FUNCTION_BLOCK PUBLIC MoveMoverToPositionZoned EXTENDS MoveMoverToPosition
VAR_INPUT
END_VAR
VAR_OUTPUT
END_VAR
VAR
	StartZone: INT;
	CurrentZone : INT;
	ZoneTransitionPositions : ARRAY[1..4] OF LREAL;
	ZoneVelocities : ARRAY[1..4] OF MC_LREAL;
END_VAR

METHOD Cycle : BOOL
VAR_INPUT
END_VAR
CASE State OF
	0:
		IF _MoveMover THEN
			_done := FALSE;
			_error := FALSE;
			_busy := TRUE;
			moveAbs.Execute := TRUE;
			StartZone := GetZone();
			moveAbs.Velocity := ZoneVelocities[StartZone];
			IF moveAbs.Busy THEN
				State := 10;
				_MoveMover := FALSE;
			END_IF
		END_IF
	
	10:
		IF NOT moveAbs.Busy THEN
			IF moveAbs.Done THEN
				_done := TRUE;
			ELSIF moveAbs.Error THEN
				_error := TRUE;
			END_IF
			_busy := FALSE;
			moveAbs.Execute := FALSE;
			State := 0;
		ELSE
			CurrentZone := GetZone();
			IF CurrentZone <> StartZone THEN
				moveAbs.Execute := FALSE;
				State := 0;
				_MoveMover := TRUE;
			END_IF
		END_IF
END_CASE

moveAbs(Axis := _axis);
END_METHOD

METHOD FB_init : BOOL
VAR_INPUT
	bInitRetains : BOOL; // if TRUE, the retain variables are initialized (warm start / cold start)
	bInCopyCode : BOOL;  // if TRUE, the instance afterwards gets moved into the copy code (online change)
	axis : REFERENCE TO AXIS_REF;
	arrPositions : ARRAY[1..4] OF LREAL;
	arrVelos : ARRAY[1..4] OF MC_LREAL;
END_VAR
SUPER^();
ZoneTransitionPositions := arrPositions;
ZoneVelocities := arrVelos;
END_METHOD

METHOD GetZone : int
VAR_INPUT
END_VAR
IF _axis.NcToPlc.ModuloActPos > ZoneTransitionPositions[1] AND _axis.NcToPlc.ModuloActPos < ZoneTransitionPositions[2] THEN
	GetZone := 1;
ELSIF (_axis.NcToPlc.ModuloActPos > ZoneTransitionPositions[2] AND _axis.NcToPlc.ModuloActPos < 11000.0) 
		OR _axis.NcToPlc.ModuloActPos > 0.0 AND  _axis.NcToPlc.ModuloActPos < ZoneTransitionPositions[3] THEN
	GetZone := 2;
ELSIF _axis.NcToPlc.ModuloActPos > ZoneTransitionPositions[3] AND _axis.NcToPlc.ModuloActPos < ZoneTransitionPositions[4] THEN
	GetZone := 3;
ELSIF _axis.NcToPlc.ModuloActPos > ZoneTransitionPositions[4] THEN
	GetZone := 4;
ELSE
	GetZone := 4;
END_IF
END_METHOD

END_FUNCTION_BLOCK

(* stored: Version 1.1.0.1, ProductVersion 3.1.4024.12
   POU MoveMoverToPositionZoned: Id {6436bcc4-2ff7-4339-a8a4-ed62d13913c2}, SpecialFunc None
   Method Cycle: Id {eb845f59-8ed2-4dab-ae31-28a22edc164c}
   Method FB_init: Id {da0f4d0e-d988-4a2c-b0bd-f2bd7411d8b3}
   Method GetZone: Id {5251f492-7e09-414e-a40c-1d2711034b00} *)
